(* PLC project Programme MGS_2-07_refactorJOY.project, CODESYS CODESYS V3.5 SP19 Patch 1 *)
(* stored: creationDateTime 2026-06-29T23:37:41.1214889, modificationDateTime 2026-06-29T22:49:33.424 *)

FUNCTION_BLOCK FB_Encoder_Safety
  VAR_INPUT
    RawSpeed : INT;  (* Vitesse brute du bus (%IW6) *)
    MaxSpeedLimit : INT;  (* Seuil critique de survitesse (en pts de vitesse) *)
    SpeedFilterTime : TIME := TIME#100ms;
    CycleTimeS : REAL;
  END_VAR
  VAR_OUTPUT
    OverspeedTrip : BOOL;  (* Ordre d'arrêt d'urgence / Freinage d'urgence *)
    FilteredSpeed : REAL;  (* Vitesse lissée pour monitoring IHM *)
  END_VAR
  VAR
    Filter : FB_Filter_PT1;  (* Réutilisation du filtre POO *)
  END_VAR

            // 1. Filtrage de la vitesse brute pour éviter les déclenchements intempestifs sur pic de com
Filter(ValueIn := INT_TO_REAL(RawSpeed), TimeConst := SpeedFilterTime, CycleTimeS := CycleTimeS);
FilteredSpeed := Filter.ValueOut;

// 2. Surveillance du seuil critique (survitesse positive ou négative)
IF ABS(FilteredSpeed) >= INT_TO_REAL(MaxSpeedLimit) THEN
    OverspeedTrip := TRUE; // Interlock / Trip à verrouiller dans votre sécurité machine
ELSE
    OverspeedTrip := FALSE;
END_IF
          
END_FUNCTION_BLOCK
